FUNCTION_BLOCK Adder
VAR_INPUT
END_VAR
VAR_OUTPUT
END_VAR
VAR
END_VAR

METHOD AddInt : INT
VAR_INPUT
  value1 : INT;
  value2 : INT;
END_VAR
AddInt := value1 + value2;
END_METHOD

END_FUNCTION_BLOCK

(* stored: Version 1.1.0.1, ProductVersion 3.1.4024.12
   POU Adder: Id {9645f133-568f-4921-a679-3f6856052c36}, SpecialFunc None
   Method AddInt: Id {072953dd-cf38-4c53-92e6-6443d1206026} *)
